TYPE "LubrValve_Alr"
VERSION : 0.1
// Block: LubrValve_Alr
   STRUCT
      CycleFeedback : Bool;
      ConnectorNotPlugged : Bool;
      ConfigError : Bool;
   END_STRUCT;

END_TYPE
